FUNCTION proj1_TupleStruct_1: LREAL
VAR_INPUT
    tuple: TupleStruct_1;
END_VAR


        proj1_TupleStruct_1 := tuple.field1;

END_FUNCTION

(* stored: ProductVersion 3.1.0.18, Version 1.1.0.1 *)
